// TIA Portal project "FactoryIO_Template_S7-1200_V15_V15.1" (V15.1)
// Vorlageprojekt für das Buch mit Zielsystem S7-1200

(* hardware
DEVICE "S7-1200-Station_1"  S7-1200 Station
   slot 0: "Baugruppenträger_0"  Rack  V1.0
   slot 1: "PLC_1"  CPU 1211C DC/DC/DC  6ES7 211-1AE40-0XB0  V4.1
*)

// ===== PLC "PLC_1"  CPU 1211C DC/DC/DC =====

VAR_GLOBAL   // PLC tag table "Standard-Variablentabelle"
   "Tag_1" AT %A0.0 : Bool;
   "Tag_2" AT %E0.0 : Bool;
   "Tag_3" AT %E0.1 : Bool;
   "Tag_4" AT %ID30 : DWord;
   "Tag_5" AT %IW32 : Word;
   "Tag_6" AT %IW36 : Int;
   "Tag_7" AT %IW40 : Int;
   "Tag_8" AT %IW30 : Int;
END_VAR

DATA_BLOCK "ExchangeData"   // DB1
{ S7_Optimized_Access := 'FALSE' }
VERSION : 0.1
   VAR
      iT1_LVL : Int;   // Poziom wody w zbiorniku 1
      iT1_DIS_FL : Int;   // Przepływ na wylocie zbiornika 1
      iT1_SP : Int;   // Wartość zadana regulacji w zbiorniku 1
      rT1_MV : Real;   // Wartość sterowania dla zbiornika 1
      rT1_H_REG : Real;   // Szerokość strefy histerezy regulatora zbiornika 1
      rT1_B_REG : Real;   // Wzmocnienie przekaźnika (Zbiornik 1)
      xT1_HH_ALM : Bool;   // Alarm poziomu HH Zbiornik 1
      xT1_H_ALM : Bool;   // Alarm poziomu H Zbiornik 1
      xT1_L_ALM : Bool;   // Alarm poziomu L Zbiornik 1
      xT1_LL_ALM : Bool;   // Alarm poziomu LL Zbiornik 1
      xT1_VLV_ALM : Bool;   // Alarm – awaria zaworu Zbiornik 1
      iT2_LVL : Int;   // Poziom wody w zbiorniku 2
      iT2_DIS_FL : Int;   // Przepływ na wylocie zbiornika 2
      iT2_SP : Int;   // Wartość zadana regulacji w zbiorniku 2
      rT2_MV : Real;   // Wartość sterowania dla zbiornika 2
      rT2_P_REG : Real;   // Wzmocnienie regulatora Zbiornik 2
      rT2_I_REG : Real;   // Parametr I regulatora Zbiornik 2
      rT2_D_REG : Real;   // Parametr D regulatora Zbiornik 2
      xT2_HH_ALM : Bool;   // Alarm poziomu HH Zbiornik 2
      xT2_H_ALM : Bool;   // Alarm poziomu H Zbiornik 2
      xT2_L_ALM : Bool;   // Alarm poziomu L Zbiornik 2
      xT2_LL_ALM : Bool;   // Alarm poziomu LL Zbiornik 2
      xT2_VLV_ALM : Bool;   // Alarm – awaria zaworu Zbiornik 2
      iT3_LVL : Int;   // Poziom wody w zbiorniku 3
      iT3_DIS_FL : Int;   // Przepływ na wylocie zbiornika 3
      iT3_SP : Int;   // Wartość zadana regulacji w zbiorniku 3
      rT3_MV : Real;   // Wartość sterowania dla zbiornika 3
      rT3_P_REG : Real;   // Wzmocnienie regulatora Zbiornik 3
      rT3_I_REG : Real;   // Parametr I regulatora Zbiornik 3
      rT3_B_REG : Real;   // Wzmocnienie przekaźnika Zbiornik 3
      xT3_HH_ALM : Bool;   // Alarm poziomu HH Zbiornik 3
      xT3_H_ALM : Bool;   // Alarm poziomu H Zbiornik 3
      xT3_L_ALM : Bool;   // Alarm poziomu L Zbiornik 3
      xT3_LL_ALM : Bool;   // Alarm poziomu LL Zbiornik 3
      xT3_VLV_ALM : Bool;   // Alarm – awaria zaworu Zbiornik 3
   END_VAR
BEGIN
END_DATA_BLOCK

FUNCTION "MHJ-PLC-Lab-Function-S71200" : Void   // FC9000, SCL
{ S7_Optimized_Access := 'TRUE' }
VERSION : 0.1
   VAR_TEMP
      rdTimeReturn : Int;
      outputTime : DTL;
      SyncVal : Byte;
      forVal : Int;
      forVal_2 : Int;
      Value : Byte;
   END_VAR
   VAR CONSTANT
      CompVal : Byte := 16#34;
      Value_01 : Byte := 16#11;
      Value_01_DW : DWord := 16#A165_D992;
      Value_02_DW : DWord := 16#58BE_4401;
   END_VAR
BEGIN

   #Value:=PEEK(area := 16#82,
        dbNumber := 0,
        byteOffset := 511);
   #Value := #Value + 1;

   POKE(area := 16#82,
        dbNumber := 0,
        byteOffset := 511,
        value := #Value);

   POKE(area:=16#81,
        dbNumber:=0,
        byteOffset:=1016,
        value:=#Value_01_DW);
   POKE(area := 16#81,
        dbNumber := 0,
        byteOffset := 1020,
        value := #Value_02_DW);

   POKE(area := 16#81,
        dbNumber := 0,
        byteOffset := 511,
        value := B#16#00);

   FOR #forVal := 0 TO 120 DO
       FOR #forVal_2:=0 TO 10 DO
           #rdTimeReturn:=RD_SYS_T(#outputTime);
           #rdTimeReturn := WR_SYS_T(#outputTime);
           #rdTimeReturn := RD_SYS_T(#outputTime);
           #rdTimeReturn := WR_SYS_T(#outputTime);
       END_FOR;
       #SyncVal:= PEEK(area := 16#81,
                      dbNumber := 0,
                      byteOffset := 511);
       IF #SyncVal = #CompVal THEN
          GOTO M_1;
       END_IF;
   END_FOR;
   RETURN;

   M_1:
   POKE(area := 16#81,
        dbNumber := 0,
        byteOffset := 511,
        value := B#16#0);
END_FUNCTION

ORGANIZATION_BLOCK "Main"   // OB1, LAD, ProgramCycle
TITLE = "Main Program Sweep (Cycle)"
{ S7_Optimized_Access := 'TRUE' }
VERSION : 0.1
   VAR_INPUT
      Initial_Call : Bool;   // Initial call of this OB
      Remanence : Bool;   // =True, if remanent data are available
   END_VAR
BEGIN

REGION Network 1: Konnektierungsbaustein für PLC-Lab
   // Im Netzwerk 1 wird der Konnektierungsbaustein für PLC-Lab aufgerufen.
   // Dieser Aufruf darf nicht entfernt werden!
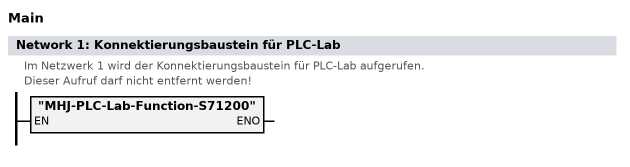
   RUNG wire#powerrail
      "MHJ-PLC-Lab-Function-S71200"()
   END_RUNG
   // the same network as SCL:
   "MHJ-PLC-Lab-Function-S71200"();
END_REGION

REGION Network 2: Ihr Programm
   // Schreiben Sie ab Netzwerk 2 Ihr Programm
END_REGION
END_ORGANIZATION_BLOCK